VAR_GLOBAL
	fbLogList : FB_Logging;
END_VAR

(* stored: Version 1.1.0.1, ProductVersion 3.1.4022.16
   GVL GVL_System: Id {b559e12f-fba4-47c6-aada-08bb316f5b43} *)
